AssertTrue(
    Condition := fb.sts.clampedHigh,
    Message   := 'Raw above rawMax must set clampedHigh');
AssertTrue(
    Condition := fb.sts.clampActive,
    Message   := 'clampActive must be TRUE when clampedHigh is set');
AssertTrue(
    Condition := ABS(fb.sts.value - 100.0) < TOL,
    Message   := 'Clamped-high output must pin to euMax (100 %)');

TEST_FINISHED();
END_METHOD

METHOD ClampPromotesGoodQualityToClamped
VAR
    fb : TcForge.FB_AnalogInput;
END_VAR
TEST('ClampPromotesGoodQualityToClamped');

// When the raw input is clamping *and* inpQuality = GOOD, the FB must
// promote quality to CLAMPED to signal "reading is legal but pinned".
fb.inRaw.nInt := -1;
fb(inpQuality := TcForge.E_IO_Quality.GOOD);

AssertTrue(
    Condition := fb.sts.clampActive,
    Message   := 'Precondition: clampActive must be TRUE');
AssertEquals_DINT(
    Expected := TO_DINT(TcForge.E_IO_Quality.CLAMPED),
    Actual   := TO_DINT(fb.sts.quality),
    Message  := 'GOOD quality must be promoted to CLAMPED while clamping');

TEST_FINISHED();
END_METHOD

METHOD ClampAsFaultRaisesClampLow
VAR
    fb : TcForge.FB_AnalogInput;
END_VAR
TEST('ClampAsFaultRaisesClampLow');

fb.cfg.clampAsFault := TRUE;
fb.inRaw.nInt := -10;
fb(inpQuality := TcForge.E_IO_Quality.GOOD);

AssertTrue(
    Condition := fb.sts.header.faulted,
    Message   := 'clampAsFault + raw below RawMin must fault the device');
AssertEquals_DINT(
    Expected := TcForge.E_AnalogInput_Fault.ClampLow,
    Actual   := fb.sts.header.faultCode,
    Message  := 'Fault code must be ClampLow');

TEST_FINISHED();
END_METHOD

METHOD ClampAsFaultRaisesClampHigh
VAR
    fb : TcForge.FB_AnalogInput;
END_VAR
TEST('ClampAsFaultRaisesClampHigh');

fb.cfg.clampAsFault := TRUE;
fb.cfg.inputType    := __SYSTEM.TYPE_CLASS.TYPE_REAL;
fb.inRaw.fReal := 50000.0;
fb(inpQuality := TcForge.E_IO_Quality.GOOD);

AssertTrue(
    Condition := fb.sts.header.faulted,
    Message   := 'clampAsFault + raw above RawMax must fault the device');
AssertEquals_DINT(
    Expected := TcForge.E_AnalogInput_Fault.ClampHigh,
    Actual   := fb.sts.header.faultCode,
    Message  := 'Fault code must be ClampHigh');

TEST_FINISHED();
END_METHOD

METHOD BadConfigRaisesFaultOnFirstScan
VAR
    fb : TcForge.FB_AnalogInput;
END_VAR
TEST('BadConfigRaisesFaultOnFirstScan');

// BadConfig check runs once on the first scan. Set rawMin >= rawMax
// BEFORE the first cyclic call so the validation can latch _configBad.
fb.cfg.rawMin := 100.0;
fb.cfg.rawMax := 100.0;
fb(inpQuality := TcForge.E_IO_Quality.GOOD);

AssertTrue(
    Condition := fb.sts.header.faulted,
    Message   := 'rawMin >= rawMax must fault the device as BadConfig');
AssertEquals_DINT(
    Expected := TcForge.E_AnalogInput_Fault.BadConfig,
    Actual   := fb.sts.header.faultCode,
    Message  := 'Fault code must be BadConfig');

TEST_FINISHED();
END_METHOD

METHOD BadQualityHoldsLastRawReading
VAR
    fb          : TcForge.FB_AnalogInput;
    snapshotRaw : REAL;
END_VAR
TEST('BadQualityHoldsLastRawReading');

// Establish a good reading first.
fb.inRaw.nInt := 10000;
fb(inpQuality := TcForge.E_IO_Quality.GOOD);
snapshotRaw := fb.sts.rawReal;

// Flip quality to BAD and change the raw wire. The FB must discard the
// fresh value and hold the last-known-good raw reading.
fb.inRaw.nInt := 25000;
fb(inpQuality := TcForge.E_IO_Quality.BAD);

AssertTrue(
    Condition := ABS(fb.sts.rawReal - snapshotRaw) < TOL,
    Message   := 'BAD quality must hold rawReal at the last-known-good value');

TEST_FINISHED();
END_METHOD

METHOD InputTypeRealReadsRealMemberOfUnion
VAR
    fb : TcForge.FB_AnalogInput;
END_VAR
TEST('InputTypeRealReadsRealMemberOfUnion');

// Select the REAL UNION member and reconfigure scaling so raw == EU,
// then confirm the FB reads the REAL alias rather than some other
// reinterpretation of the same bytes.
fb.cfg.inputType := __SYSTEM.TYPE_CLASS.TYPE_REAL;
fb.cfg.rawMin    := 0.0;
fb.cfg.rawMax    := 100.0;
fb.cfg.euMin     := 0.0;
fb.cfg.euMax     := 100.0;

fb.inRaw.fReal := 42.5;
fb(inpQuality := TcForge.E_IO_Quality.GOOD);

AssertTrue(
    Condition := ABS(fb.sts.rawReal - 42.5) < TOL,
    Message   := 'TYPE_REAL must read inRaw.fReal directly into rawReal');
AssertTrue(
    Condition := ABS(fb.sts.value - 42.5) < TOL,
    Message   := 'Identity scaling must leave value equal to the raw REAL input');

TEST_FINISHED();
END_METHOD

METHOD QualityTagPropagatesToStatus
VAR
    fb : TcForge.FB_AnalogInput;
END_VAR
TEST('QualityTagPropagatesToStatus');

// The FB must echo inpQuality into sts.quality each cycle (subject to
// the clamp promotion covered by ClampPromotesGoodQualityToClamped).
fb.inRaw.nInt := 10000;
fb(inpQuality := TcForge.E_IO_Quality.GOOD);
AssertEquals_DINT(
    Expected := TO_DINT(TcForge.E_IO_Quality.GOOD),
    Actual   := TO_DINT(fb.sts.quality),
    Message  := 'quality must mirror inpQuality = GOOD when not clamping');

fb(inpQuality := TcForge.E_IO_Quality.UNKNOWN);
AssertEquals_DINT(
    Expected := TO_DINT(TcForge.E_IO_Quality.UNKNOWN),
    Actual   := TO_DINT(fb.sts.quality),
    Message  := 'quality must mirror inpQuality = UNKNOWN');

fb(inpQuality := TcForge.E_IO_Quality.BAD);
AssertEquals_DINT(
    Expected := TO_DINT(TcForge.E_IO_Quality.BAD),
    Actual   := TO_DINT(fb.sts.quality),
    Message  := 'quality must mirror inpQuality = BAD');

TEST_FINISHED();
END_METHOD

END_FUNCTION_BLOCK

// ---- Tests/FB_AnalogOutput_Test.TcPOU
// Tests exercise the public input/output and command contracts.
FUNCTION_BLOCK FB_AnalogOutput_Test EXTENDS TcUnit.FB_TestSuite
VAR CONSTANT
    TOL     : REAL := 1E-3;
    RAW_TOL : INT  := 1;
END_VAR

InitialStatusPublishesDefaults();
LinearScalingMapsEndpointsAndMidpoint();
ClampHighPinsCommandAndFlagsClampedHigh();
ClampLowPinsCommandAndFlagsClampedLow();
CommandedEchoesUnclampedRequest();
RawBypassSkipsClampAndScaling();
ClampAsFaultRaisesClampHigh();
ClampAsFaultRaisesClampLow();
BadConfigRaisesFaultOnFirstScan();
OutputTypeRealWritesRealUnionMember();
BadQualityHoldsLastWrittenUnion();
QualityTagPropagatesToStatus();
SetValueRejectedWhenSourceLockedToProg();
SetValueAcceptedFromProgWhenLocked();

METHOD InitialStatusPublishesDefaults
VAR
    fb : TcForge.FB_AnalogOutput;
END_VAR
TEST('InitialStatusPublishesDefaults');

// Default cfg: INT terminal, EU 0..100 % scaled into raw 0..32767,
// clampAsFault disabled. Before any SetValue the persistent command is
// zero, so the FB must publish a clean zero command with no clamp
// flags and no fault.
fb(inpQuality := TcForge.E_IO_Quality.GOOD);

AssertTrue(
    Condition := ABS(fb.sts.value) < TOL,
    Message   := 'Fresh instance must publish value = 0 for an unset command');
AssertTrue(
    Condition := ABS(fb.sts.commanded) < TOL,
    Message   := 'Fresh instance must publish commanded = 0');
AssertTrue(
    Condition := ABS(fb.sts.rawReal) < TOL,
    Message   := 'Fresh instance must publish rawReal = 0');
AssertFalse(
    Condition := fb.sts.clampActive,
    Message   := 'Zero command is inside [minCv, maxCv] so clampActive must be FALSE');
AssertFalse(
    Condition := fb.sts.header.faulted,
    Message   := 'Default cfg is valid so the first scan must not fault');

TEST_FINISHED();
END_METHOD

METHOD LinearScalingMapsEndpointsAndMidpoint
VAR
    fb  : TcForge.FB_AnalogOutput;
    rsp : TcForge.E_RpcMethodResponse;
END_VAR
TEST('LinearScalingMapsEndpointsAndMidpoint');

// Default cfg: EU 0..100 -> raw 0..32767. Verify the two endpoints and
// the midpoint land where the linear recurrence says they should,
// both in sts.rawReal (REAL) and in outRaw.nInt (after INT coercion).
//
//     rawReal = rawMin + (cmd - euMin)
//                             * (rawMax - rawMin)
//                             / (euMax - euMin)

rsp := fb.SetValue(rValue := 0.0);
fb(inpQuality := TcForge.E_IO_Quality.GOOD);
AssertTrue(
    Condition := ABS(fb.sts.rawReal - 0.0) < TOL,
    Message   := 'cmd = euMin must map to rawMin (0)');
AssertTrue(
    Condition := ABS(fb.outRaw.nInt) <= RAW_TOL,
    Message   := 'UNION INT alias must receive ~0 for a 0 %% command');

rsp := fb.SetValue(rValue := 100.0);
fb(inpQuality := TcForge.E_IO_Quality.GOOD);
AssertTrue(
    Condition := ABS(fb.sts.rawReal - 32767.0) < TOL,
    Message   := 'cmd = euMax must map to rawMax (32767)');
AssertTrue(
    Condition := ABS(fb.outRaw.nInt - 32767) <= RAW_TOL,
    Message   := 'UNION INT alias must receive ~32767 for a 100 %% command');

rsp := fb.SetValue(rValue := 50.0);
fb(inpQuality := TcForge.E_IO_Quality.GOOD);
AssertTrue(
    Condition := ABS(fb.sts.rawReal - 16383.5) < 0.01,
    Message   := 'cmd at midpoint must map to raw midpoint');
AssertTrue(
    Condition := ABS(fb.outRaw.nInt - 16384) <= RAW_TOL,
    Message   := 'UNION INT alias must receive the rounded midpoint raw');

TEST_FINISHED();
END_METHOD

METHOD ClampHighPinsCommandAndFlagsClampedHigh
VAR
    fb  : TcForge.FB_AnalogOutput;
    rsp : TcForge.E_RpcMethodResponse;
END_VAR
TEST('ClampHighPinsCommandAndFlagsClampedHigh');

// Drive a command above maxCv. clampedHigh must fire, clampActive must
// track, value must pin at maxCv, and the raw write must use the
// pinned value — not the unclamped request.
rsp := fb.SetValue(rValue := 150.0);
fb(inpQuality := TcForge.E_IO_Quality.GOOD);

AssertTrue(
    Condition := fb.sts.clampedHigh,
    Message   := 'cmd above maxCv must set clampedHigh');
AssertTrue(
    Condition := fb.sts.clampActive,
    Message   := 'clampActive must be TRUE whenever either clamp direction is active');
AssertTrue(
    Condition := ABS(fb.sts.value - 100.0) < TOL,
    Message   := 'value must pin at maxCv (100 %%) when clamping high');
AssertTrue(
    Condition := ABS(fb.sts.rawReal - 32767.0) < TOL,
    Message   := 'rawReal must reflect the clamped EU, not the unclamped request');
AssertFalse(
    Condition := fb.sts.header.faulted,
    Message   := 'clampAsFault = FALSE by default; clamp alone must not fault the device');

TEST_FINISHED();
END_METHOD

METHOD ClampLowPinsCommandAndFlagsClampedLow
VAR
    fb  : TcForge.FB_AnalogOutput;
    rsp : TcForge.E_RpcMethodResponse;
END_VAR
TEST('ClampLowPinsCommandAndFlagsClampedLow');

// Drive a command below minCv. clampedLow must fire, value must pin
// at minCv, raw write uses the pinned value.
rsp := fb.SetValue(rValue := -25.0);
fb(inpQuality := TcForge.E_IO_Quality.GOOD);

AssertTrue(
    Condition := fb.sts.clampedLow,
    Message   := 'cmd below minCv must set clampedLow');
AssertTrue(
    Condition := fb.sts.clampActive,
    Message   := 'clampActive must be TRUE whenever either clamp direction is active');
AssertTrue(
    Condition := ABS(fb.sts.value - 0.0) < TOL,
    Message   := 'value must pin at minCv (0 %%) when clamping low');
AssertTrue(
    Condition := ABS(fb.sts.rawReal - 0.0) < TOL,
    Message   := 'rawReal must reflect the clamped EU, not the unclamped request');
AssertFalse(
    Condition := fb.sts.header.faulted,
    Message   := 'clampAsFault = FALSE by default; clamp alone must not fault the device');

TEST_FINISHED();
END_METHOD

METHOD CommandedEchoesUnclampedRequest
VAR
    fb  : TcForge.FB_AnalogOutput;
    rsp : TcForge.E_RpcMethodResponse;
END_VAR
TEST('CommandedEchoesUnclampedRequest');

// sts.commanded publishes the pre-clamp request; restart restoration is separately qualified
// via _requestSync. The tests above already prove sts.value tracks the
// clamped write; here we pin down that sts.commanded preserves the
// operator's original intent so the HMI can show "you asked for 150,
// we clamped to 100".
rsp := fb.SetValue(rValue := 150.0);
fb(inpQuality := TcForge.E_IO_Quality.GOOD);

AssertTrue(
    Condition := ABS(fb.sts.commanded - 150.0) < TOL,
    Message   := 'commanded must echo the unclamped SetValue input');
AssertTrue(
    Condition := ABS(fb.sts.value - 100.0) < TOL,
    Message   := 'value must be the clamped command actually written');

rsp := fb.SetValue(rValue := -7.5);
fb(inpQuality := TcForge.E_IO_Quality.GOOD);

AssertTrue(
    Condition := ABS(fb.sts.commanded - (-7.5)) < TOL,
    Message   := 'commanded must echo a negative request even when clamped low');
AssertTrue(
    Condition := ABS(fb.sts.value - 0.0) < TOL,
    Message   := 'value must pin at minCv under a low clamp');

TEST_FINISHED();
END_METHOD

METHOD RawBypassSkipsClampAndScaling
VAR
    fb  : TcForge.FB_AnalogOutput;
    rsp : TcForge.E_RpcMethodResponse;
END_VAR
TEST('RawBypassSkipsClampAndScaling');

// useRawValue = TRUE writes the command REAL straight into the UNION
// without clamping, so a 12345 command lands as 12345 on the raw INT
// alias even though that is well above maxCv and well above rawMax.
fb.cfg.useRawValue := TRUE;
rsp := fb.SetValue(rValue := 12345.0);
fb(inpQuality := TcForge.E_IO_Quality.GOOD);

AssertTrue(
    Condition := ABS(fb.sts.rawReal - 12345.0) < TOL,
    Message   := 'With useRawValue = TRUE, rawReal must equal the raw command');
AssertTrue(
    Condition := ABS(fb.sts.value - 12345.0) < TOL,
    Message   := 'With useRawValue = TRUE, value must equal the raw command');
AssertFalse(
    Condition := fb.sts.clampedLow,
    Message   := 'Raw bypass must not flag clampedLow');
AssertFalse(
    Condition := fb.sts.clampedHigh,
    Message   := 'Raw bypass must not flag clampedHigh');
AssertFalse(
    Condition := fb.sts.clampActive,
    Message   := 'Raw bypass must not flag clampActive');
AssertTrue(
    Condition := ABS(fb.outRaw.nInt - 12345) <= RAW_TOL,
    Message   := 'UNION INT alias must receive the raw command unchanged');

TEST_FINISHED();
END_METHOD

METHOD ClampAsFaultRaisesClampHigh
VAR
    fb  : TcForge.FB_AnalogOutput;
    rsp : TcForge.E_RpcMethodResponse;
END_VAR
TEST('ClampAsFaultRaisesClampHigh');

fb.cfg.clampAsFault := TRUE;
rsp := fb.SetValue(rValue := 150.0);
fb(inpQuality := TcForge.E_IO_Quality.GOOD);

AssertTrue(
    Condition := fb.sts.header.faulted,
    Message   := 'clampAsFault + cmd above maxCv must fault the device');
AssertEquals_DINT(
    Expected := TcForge.E_AnalogOutput_Fault.ClampHigh,
    Actual   := fb.sts.header.faultCode,
    Message  := 'Fault code must be ClampHigh');

TEST_FINISHED();
END_METHOD

METHOD ClampAsFaultRaisesClampLow
VAR
    fb  : TcForge.FB_AnalogOutput;
    rsp : TcForge.E_RpcMethodResponse;
END_VAR
TEST('ClampAsFaultRaisesClampLow');

fb.cfg.clampAsFault := TRUE;
rsp := fb.SetValue(rValue := -5.0);
fb(inpQuality := TcForge.E_IO_Quality.GOOD);

AssertTrue(
    Condition := fb.sts.header.faulted,
    Message   := 'clampAsFault + cmd below minCv must fault the device');
AssertEquals_DINT(
    Expected := TcForge.E_AnalogOutput_Fault.ClampLow,
    Actual   := fb.sts.header.faultCode,
    Message  := 'Fault code must be ClampLow');

TEST_FINISHED();
END_METHOD

METHOD BadConfigRaisesFaultOnFirstScan
VAR
    fb : TcForge.FB_AnalogOutput;
END_VAR
TEST('BadConfigRaisesFaultOnFirstScan');

// BadConfig check runs once on the first scan. Set rawMin > rawMax
// BEFORE the first cyclic call so the validation can latch _configBad.
fb.cfg.rawMin := 200.0;
fb.cfg.rawMax := 100.0;
fb(inpQuality := TcForge.E_IO_Quality.GOOD);

AssertTrue(
    Condition := fb.sts.header.faulted,
    Message   := 'rawMin > rawMax must fault the device as BadConfig');
AssertEquals_DINT(
    Expected := TcForge.E_AnalogOutput_Fault.BadConfig,
    Actual   := fb.sts.header.faultCode,
    Message  := 'Fault code must be BadConfig');

TEST_FINISHED();
END_METHOD

METHOD OutputTypeRealWritesRealUnionMember
VAR
    fb  : TcForge.FB_AnalogOutput;
    rsp : TcForge.E_RpcMethodResponse;
END_VAR
TEST('OutputTypeRealWritesRealUnionMember');

// Select the REAL UNION member and reconfigure scaling so raw == EU,
// then confirm the FB writes the REAL alias with the exact command
// (no integer coercion).
fb.cfg.outputType := __SYSTEM.TYPE_CLASS.TYPE_REAL;
fb.cfg.rawMin     := 0.0;
fb.cfg.rawMax     := 100.0;
fb.cfg.euMin      := 0.0;
fb.cfg.euMax      := 100.0;

rsp := fb.SetValue(rValue := 42.5);
fb(inpQuality := TcForge.E_IO_Quality.GOOD);

AssertTrue(
    Condition := ABS(fb.sts.rawReal - 42.5) < TOL,
    Message   := 'Identity scaling must leave rawReal equal to the command');
AssertTrue(
    Condition := ABS(fb.outRaw.fReal - 42.5) < TOL,
    Message   := 'TYPE_REAL must write outRaw.fReal directly with the command');

TEST_FINISHED();
END_METHOD

METHOD BadQualityHoldsLastWrittenUnion
VAR
    fb           : TcForge.FB_AnalogOutput;
    rsp          : TcForge.E_RpcMethodResponse;
    snapshot     : DWORD;
END_VAR
TEST('BadQualityHoldsLastWrittenUnion');
fb.cfg.holdOnBadQuality := TRUE;

// Establish a known value in the UNION under GOOD quality.
rsp := fb.SetValue(rValue := 25.0);
fb(inpQuality := TcForge.E_IO_Quality.GOOD);
snapshot := fb.outRaw.dw;

// Flip quality to BAD and change the commanded value. The FB must
// still recompute sts.rawReal (it is pure output of the pipeline),
// but it must NOT touch the hardware-linked UNION — the terminal
// keeps its last-known-good bytes.
rsp := fb.SetValue(rValue := 75.0);
fb(inpQuality := TcForge.E_IO_Quality.BAD);

AssertEquals_DWORD(
    Expected := snapshot,
    Actual   := fb.outRaw.dw,
    Message  := 'BAD quality must skip the UNION write and hold the last-known-good bytes');

TEST_FINISHED();
END_METHOD

METHOD QualityTagPropagatesToStatus
VAR
    fb : TcForge.FB_AnalogOutput;
END_VAR
TEST('QualityTagPropagatesToStatus');

// FB_AnalogOutput echoes inpQuality straight through (no clamp-to-CLAMPED
// promotion like the input FB does — output-side consumers treat CLAMPED
// as informational and the write still goes out).
fb(inpQuality := TcForge.E_IO_Quality.GOOD);
AssertEquals_DINT(
    Expected := TO_DINT(TcForge.E_IO_Quality.GOOD),
    Actual   := TO_DINT(fb.sts.quality),
    Message  := 'quality must mirror inpQuality = GOOD');

fb(inpQuality := TcForge.E_IO_Quality.UNKNOWN);
AssertEquals_DINT(
    Expected := TO_DINT(TcForge.E_IO_Quality.UNKNOWN),
    Actual   := TO_DINT(fb.sts.quality),
    Message  := 'quality must mirror inpQuality = UNKNOWN');

fb(inpQuality := TcForge.E_IO_Quality.BAD);
AssertEquals_DINT(
    Expected := TO_DINT(TcForge.E_IO_Quality.BAD),
    Actual   := TO_DINT(fb.sts.quality),
    Message  := 'quality must mirror inpQuality = BAD');

TEST_FINISHED();
END_METHOD

METHOD SetValueRejectedWhenSourceLockedToProg
VAR
    fb  : TcForge.FB_AnalogOutput;
    rsp : TcForge.E_RpcMethodResponse;
END_VAR
TEST('SetValueRejectedWhenSourceLockedToProg');

// With source locked to PROG, an OPERATOR SetValue must be rejected
// with SOURCE_LOCKED, the persistent command must stay at zero, and
// no clamp flags or writes may trigger.
fb.LockSource(bLock := TRUE);

rsp := fb.SetValue(rValue := 42.0, eRequester := TcForge.E_Requester.OPERATOR);
fb(inpQuality := TcForge.E_IO_Quality.GOOD);

AssertEquals_DINT(
    Expected := TO_DINT(TcForge.E_RpcMethodResponse.REJECTED_SOURCE_NOT_ALLOWED),
    Actual   := TO_DINT(rsp),
    Message  := 'OPERATOR SetValue against a source-locked FB must be rejected');
AssertTrue(
    Condition := ABS(fb.sts.commanded - 0.0) < TOL,
    Message   := 'A rejected SetValue must leave commanded unchanged');
AssertTrue(
    Condition := ABS(fb.sts.value - 0.0) < TOL,
    Message   := 'A rejected SetValue must leave value unchanged');

TEST_FINISHED();
END_METHOD

METHOD SetValueAcceptedFromProgWhenLocked
VAR
    fb  : TcForge.FB_AnalogOutput;
    rsp : TcForge.E_RpcMethodResponse;
END_VAR
TEST('SetValueAcceptedFromProgWhenLocked');

// With source locked to PROG, a PROG SetValue must still be accepted —
// that's the whole point of locking: only the program may drive.
fb.LockSource(bLock := TRUE);

rsp := fb.SetValue(rValue := 42.0, eRequester := TcForge.E_Requester.PROG);
fb(inpQuality := TcForge.E_IO_Quality.GOOD);

AssertEquals_DINT(
    Expected := TO_DINT(TcForge.E_RpcMethodResponse.ACCEPTED),
    Actual   := TO_DINT(rsp),
    Message  := 'PROG SetValue must be accepted even when source-locked to PROG');
AssertTrue(
    Condition := ABS(fb.sts.commanded - 42.0) < TOL,
    Message   := 'Accepted PROG SetValue must update commanded');
AssertTrue(
    Condition := ABS(fb.sts.value - 42.0) < TOL,
    Message   := 'Accepted PROG SetValue must flow into value');

TEST_FINISHED();
END_METHOD

END_FUNCTION_BLOCK

// ---- Tests/FB_AlarmThreshold_Test.TcPOU
// Tests for FB_AlarmThreshold. The FB itself is thin — it owns the
// direction select (bFailHigh / bFailLow) and the raw comparator, then
// forwards everything into FB_AlarmBase._Evaluate(). The shared alarm
// contract (debounce, latch/ack state machine, severity, message echo,
// source lock, disable gating) is already covered by FB_AlarmSimple_Test,
// so this suite focuses on the threshold-specific logic plus a couple of
// smoke tests that confirm the base pipeline is wired in.
FUNCTION_BLOCK FB_AlarmThreshold_Test EXTENDS TcUnit.FB_TestSuite

FailHighTripsStrictlyAboveThreshold();
FailHighIgnoresAtOrBelowThreshold();
FailLowTripsStrictlyBelowThreshold();
FailLowIgnoresAtOrAboveThreshold();
BothDirectionsAreInvalid();
NeitherDirectionIsInvalid();
DisabledSuppressesTripRegardlessOfValue();
SeverityFlowsThroughBaseOnActive();
LatchingHoldsAfterValueReturnsToSafe();
MessageEchoedFromCommonCfg();

METHOD FailHighTripsStrictlyAboveThreshold
VAR
    fb : TcForge.FB_AlarmThreshold;
END_VAR
TEST('FailHighTripsStrictlyAboveThreshold');

// bFailHigh + inpValue > fThreshold must trip the alarm. Configured as
// non-latching so we can observe the raw rollup directly.
fb.cfg.common.bEnable := TRUE;
fb.cfg.fThreshold     := 80.0;
fb.cfg.bFailHigh      := TRUE;

fb(inpValue := 80.1);
AssertTrue(
    Condition := fb.sts.active,
    Message   := 'Fail-high alarm must go active when inpValue exceeds fThreshold');
AssertTrue(
    Condition := fb.sts.raw,
    Message   := 'Fail-high rollup must mirror the strict > comparison on sts.raw');

TEST_FINISHED();
END_METHOD

METHOD FailHighIgnoresAtOrBelowThreshold
VAR
    fb : TcForge.FB_AlarmThreshold;
END_VAR
TEST('FailHighIgnoresAtOrBelowThreshold');

// inpValue == fThreshold must NOT trip a fail-high alarm: the comparison
// is a strict `>` so a reading that is exactly at the threshold is
// considered still-safe. Any inequality in the other direction is also
// ignored. Together these prevent jittery readings from chattering on
// the threshold boundary.
fb.cfg.common.bEnable := TRUE;
fb.cfg.fThreshold     := 80.0;
fb.cfg.bFailHigh      := TRUE;

fb(inpValue := 80.0);
AssertFalse(
    Condition := fb.sts.active,
    Message   := 'Fail-high must not trip when inpValue equals fThreshold (strict >)');

fb(inpValue := 10.0);
AssertFalse(
    Condition := fb.sts.active,
    Message   := 'Fail-high must not trip when inpValue is well below fThreshold');

TEST_FINISHED();
END_METHOD

METHOD FailLowTripsStrictlyBelowThreshold
VAR
    fb : TcForge.FB_AlarmThreshold;
END_VAR
TEST('FailLowTripsStrictlyBelowThreshold');

fb.cfg.common.bEnable := TRUE;
fb.cfg.fThreshold     := 10.0;
fb.cfg.bFailLow       := TRUE;

fb(inpValue := 9.9);
AssertTrue(
    Condition := fb.sts.active,
    Message   := 'Fail-low alarm must go active when inpValue falls below fThreshold');

TEST_FINISHED();
END_METHOD

METHOD FailLowIgnoresAtOrAboveThreshold
VAR
    fb : TcForge.FB_AlarmThreshold;
END_VAR
TEST('FailLowIgnoresAtOrAboveThreshold');

fb.cfg.common.bEnable := TRUE;
fb.cfg.fThreshold     := 10.0;
fb.cfg.bFailLow       := TRUE;

fb(inpValue := 10.0);
AssertFalse(
    Condition := fb.sts.active,
    Message   := 'Fail-low must not trip when inpValue equals fThreshold (strict <)');

fb(inpValue := 50.0);
AssertFalse(
    Condition := fb.sts.active,
    Message   := 'Fail-low must not trip when inpValue is well above fThreshold');

TEST_FINISHED();
END_METHOD

METHOD BothDirectionsAreInvalid
VAR
    fb : TcForge.FB_AlarmThreshold;
END_VAR
TEST('BothDirectionsAreInvalid');
fb.cfg.common.bEnable := TRUE;
fb.cfg.bFailHigh := TRUE; fb.cfg.bFailLow := TRUE;
fb(inpValue := 60.0);
AssertFalse(Condition := fb.sts.valid, Message := 'Exactly one direction is required');
AssertEquals_DINT(Expected := TcForge.E_AlarmEvaluation.InvalidConfig, Actual := fb.sts.evaluationState, Message := 'Invalid configuration is visible');
AssertFalse(Condition := fb.sts.active, Message := 'Invalid fresh configuration does not invent a trip');
TEST_FINISHED();
END_METHOD

METHOD NeitherDirectionIsInvalid
VAR
    fb : TcForge.FB_AlarmThreshold;
END_VAR
TEST('NeitherDirectionIsInvalid');
fb.cfg.common.bEnable := TRUE;
fb.cfg.bFailHigh := FALSE; fb.cfg.bFailLow := FALSE;
fb(inpValue := 60.0);
AssertFalse(Condition := fb.sts.valid, Message := 'Exactly one direction is required');
AssertEquals_DINT(Expected := TcForge.E_AlarmEvaluation.InvalidConfig, Actual := fb.sts.evaluationState, Message := 'Invalid configuration is visible');
AssertFalse(Condition := fb.sts.active, Message := 'Invalid fresh configuration does not invent a trip');
TEST_FINISHED();
END_METHOD

METHOD DisabledSuppressesTripRegardlessOfValue
VAR
    fb : TcForge.FB_AlarmThreshold;
END_VAR
TEST('DisabledSuppressesTripRegardlessOfValue');

// bEnable = FALSE shortcuts _Evaluate before the latch / severity logic
// runs. Confirm the threshold FB inherits that behaviour even when the
// raw comparison would otherwise fire.
fb.cfg.common.bEnable := FALSE;
fb.cfg.common.eSeverity := TcForge.E_AlarmSeverity.CRITICAL;
fb.cfg.fThreshold       := 50.0;
fb.cfg.bFailHigh        := TRUE;

fb(inpValue := 999.0);

AssertFalse(
    Condition := fb.sts.active,
    Message   := 'Disabled threshold alarm must not trip even with inpValue way above fThreshold');
AssertEquals_USINT(
    Expected := TcForge.E_AlarmSeverity.NONE,
    Actual   := fb.sts.eSeverity,
    Message  := 'Disabled alarm must report severity NONE regardless of value');

TEST_FINISHED();
END_METHOD

METHOD SeverityFlowsThroughBaseOnActive
VAR
    fb : TcForge.FB_AlarmThreshold;
END_VAR
TEST('SeverityFlowsThroughBaseOnActive');

// Smoke test: when the threshold condition trips, the base's severity
// propagation still runs. This proves the threshold FB does call
// _Evaluate() and does not short-circuit the pipeline.
fb.cfg.common.bEnable     := TRUE;
fb.cfg.common.bRequireAck := FALSE;
fb.cfg.common.eSeverity   := TcForge.E_AlarmSeverity.WARNING;
fb.cfg.fThreshold         := 50.0;
fb.cfg.bFailHigh          := TRUE;

fb(inpValue := 60.0);
AssertEquals_USINT(
    Expected := TcForge.E_AlarmSeverity.WARNING,
    Actual   := fb.sts.eSeverity,
    Message  := 'Active threshold alarm must publish the configured severity');

fb(inpValue := 40.0);
AssertEquals_USINT(
    Expected := TcForge.E_AlarmSeverity.NONE,
    Actual   := fb.sts.eSeverity,
    Message  := 'Cleared threshold alarm must drop severity to NONE');

TEST_FINISHED();
END_METHOD

METHOD LatchingHoldsAfterValueReturnsToSafe
VAR
    fb : TcForge.FB_AlarmThreshold;
END_VAR
TEST('LatchingHoldsAfterValueReturnsToSafe');

// Smoke test for the bRequireAck pathway through the threshold FB.
// The base FB_AlarmSimple_Test already exercises the full latch/ack
// state machine in isolation; here we just confirm the threshold FB
// keeps the latch engaged after the process value returns below the
// threshold (which is the whole reason to latch on a transient spike).
fb.cfg.common.bEnable     := TRUE;
fb.cfg.common.bRequireAck := TRUE;
fb.cfg.common.eSeverity   := TcForge.E_AlarmSeverity.CRITICAL;
fb.cfg.fThreshold         := 80.0;
fb.cfg.bFailHigh          := TRUE;

fb(inpValue := 90.0);
AssertTrue(
    Condition := fb.sts.active AND fb.sts.latched,
    Message   := 'Latching threshold alarm must go active+latched on a trip');

fb(inpValue := 50.0);
AssertTrue(
    Condition := fb.sts.active,
    Message   := 'Latched threshold alarm must stay active after inpValue returns below fThreshold');

TEST_FINISHED();
END_METHOD

METHOD MessageEchoedFromCommonCfg
VAR
    fb : TcForge.FB_AlarmThreshold;
END_VAR
TEST('MessageEchoedFromCommonCfg');

// Confirms that a threshold alarm hands the common cfg (including
// sMessage) to the base unchanged. Regression guard against future
// refactors of ST_AlarmThreshold_Cfg that might shadow `common`.
fb.cfg.common.bEnable  := TRUE;
fb.cfg.common.sMessage := 'Reactor temp > 80C';
fb.cfg.fThreshold      := 80.0;
fb.cfg.bFailHigh       := TRUE;

fb(inpValue := 50.0);

AssertEquals_STRING(
    Expected := 'Reactor temp > 80C',
    Actual   := fb.sts.sMessage,
    Message  := 'sts.sMessage must echo cfg.common.sMessage verbatim');

TEST_FINISHED();
END_METHOD

END_FUNCTION_BLOCK

// ---- Tests/FB_AlarmDeviation_Test.TcPOU
// Tests for FB_AlarmDeviation. The deviation FB owns two comparator
// modes — absolute band (fLowLimit..fHighLimit) and asymmetric setpoint
// deviation (inpSetpoint +/- limit) — and forwards the boolean rollup
// into FB_AlarmBase._Evaluate(). The shared alarm contract (debounce,
// latch/ack, severity, source lock) is already covered by
// FB_AlarmSimple_Test, so this suite focuses on the deviation-specific
// comparator logic plus a smoke test confirming the base pipeline runs.
FUNCTION_BLOCK FB_AlarmDeviation_Test EXTENDS TcUnit.FB_TestSuite

AbsoluteModeTripsAboveHighLimit();
AbsoluteModeTripsBelowLowLimit();
AbsoluteModeStaysQuietWithinBand();
AbsoluteModeIgnoresInpSetpoint();
SetpointModeTripsAbovePositiveDeviation();
SetpointModeTripsBelowNegativeDeviation();
SetpointModeTracksMovingSetpoint();
SetpointModeAllowsAsymmetricLimits();
DisabledSuppressesTripRegardlessOfValue();
SeverityFlowsThroughBaseOnActive();

METHOD AbsoluteModeTripsAboveHighLimit
VAR
    fb : TcForge.FB_AlarmDeviation;
END_VAR
TEST('AbsoluteModeTripsAboveHighLimit');

// Absolute mode: limits are direct values on inpPv (inpSetpoint ignored).
fb.cfg.common.bEnable := TRUE;
fb.cfg.bUseSetpoint   := FALSE;
fb.cfg.fHighLimit     := 95.0;
fb.cfg.fLowLimit      := 10.0;

fb(inpPv := 96.0, inpSetpoint := 0.0);

AssertTrue(
    Condition := fb.sts.active,
    Message   := 'Absolute mode must trip when inpPv is strictly above fHighLimit');

TEST_FINISHED();
END_METHOD

METHOD AbsoluteModeTripsBelowLowLimit
VAR
    fb : TcForge.FB_AlarmDeviation;
END_VAR
TEST('AbsoluteModeTripsBelowLowLimit');

fb.cfg.common.bEnable := TRUE;
fb.cfg.bUseSetpoint   := FALSE;
fb.cfg.fHighLimit     := 95.0;
fb.cfg.fLowLimit      := 10.0;

fb(inpPv := 9.0, inpSetpoint := 0.0);

AssertTrue(
    Condition := fb.sts.active,
    Message   := 'Absolute mode must trip when inpPv is strictly below fLowLimit');

TEST_FINISHED();
END_METHOD

METHOD AbsoluteModeStaysQuietWithinBand
VAR
    fb : TcForge.FB_AlarmDeviation;
END_VAR
TEST('AbsoluteModeStaysQuietWithinBand');

// Boundaries are inclusive (strict > and strict <), so exactly-at-limit
// readings must not trip. Middle-of-band must also not trip.
fb.cfg.common.bEnable := TRUE;
fb.cfg.bUseSetpoint   := FALSE;
fb.cfg.fHighLimit     := 95.0;
fb.cfg.fLowLimit      := 10.0;

fb(inpPv := 10.0);
AssertFalse(
    Condition := fb.sts.active,
    Message   := 'Absolute mode must not trip at the low boundary exactly (strict <)');

fb(inpPv := 95.0);
AssertFalse(
    Condition := fb.sts.active,
    Message   := 'Absolute mode must not trip at the high boundary exactly (strict >)');

fb(inpPv := 50.0);
AssertFalse(
    Condition := fb.sts.active,
    Message   := 'Absolute mode must not trip mid-band');

TEST_FINISHED();
END_METHOD

METHOD AbsoluteModeIgnoresInpSetpoint
VAR
    fb : TcForge.FB_AlarmDeviation;
END_VAR
TEST('AbsoluteModeIgnoresInpSetpoint');

// Absolute mode must not look at inpSetpoint at all — otherwise a drifting
// setpoint could silently shift the safe band. Same PV, different SP,
// same result.
fb.cfg.common.bEnable := TRUE;
fb.cfg.bUseSetpoint   := FALSE;
fb.cfg.fHighLimit     := 95.0;
fb.cfg.fLowLimit      := 10.0;

fb(inpPv := 50.0, inpSetpoint := 0.0);
AssertFalse(
    Condition := fb.sts.active,
    Message   := 'Absolute mode with SP=0: mid-band must stay quiet');

fb(inpPv := 50.0, inpSetpoint := 1000.0);
AssertFalse(
    Condition := fb.sts.active,
    Message   := 'Absolute mode must ignore inpSetpoint: same PV stays quiet regardless of SP');

TEST_FINISHED();
END_METHOD

METHOD SetpointModeTripsAbovePositiveDeviation
VAR
    fb : TcForge.FB_AlarmDeviation;
END_VAR
TEST('SetpointModeTripsAbovePositiveDeviation');

// Setpoint mode: fHighLimit is a +deviation from inpSetpoint.
// SP=100, +5 band => trip above 105.
fb.cfg.common.bEnable := TRUE;
fb.cfg.bUseSetpoint   := TRUE;
fb.cfg.fHighLimit     := 5.0;
fb.cfg.fLowLimit      := 5.0;

fb(inpPv := 106.0, inpSetpoint := 100.0);

AssertTrue(
    Condition := fb.sts.active,
    Message   := 'Setpoint mode must trip when inpPv exceeds inpSetpoint + fHighLimit');

TEST_FINISHED();
END_METHOD

METHOD SetpointModeTripsBelowNegativeDeviation
VAR
    fb : TcForge.FB_AlarmDeviation;
END_VAR
TEST('SetpointModeTripsBelowNegativeDeviation');

fb.cfg.common.bEnable := TRUE;
fb.cfg.bUseSetpoint   := TRUE;
fb.cfg.fHighLimit     := 5.0;
fb.cfg.fLowLimit      := 5.0;

fb(inpPv := 94.0, inpSetpoint := 100.0);

AssertTrue(
    Condition := fb.sts.active,
    Message   := 'Setpoint mode must trip when inpPv falls below inpSetpoint - fLowLimit');

TEST_FINISHED();
END_METHOD

METHOD SetpointModeTracksMovingSetpoint
VAR
    fb : TcForge.FB_AlarmDeviation;
END_VAR
TEST('SetpointModeTracksMovingSetpoint');

// Whole point of setpoint mode: the safe band follows the setpoint.
// A PV that was in-band at SP=100 must be out-of-band once SP=200 if the
// deviations are small — and back in-band when SP catches up.
fb.cfg.common.bEnable     := TRUE;
fb.cfg.common.bRequireAck := FALSE;
fb.cfg.bUseSetpoint       := TRUE;
fb.cfg.fHighLimit         := 5.0;
fb.cfg.fLowLimit          := 5.0;

// PV=100 is dead on SP=100 => safe.
fb(inpPv := 100.0, inpSetpoint := 100.0);
AssertFalse(
    Condition := fb.sts.active,
    Message   := 'PV at SP is always safe');

// SP jumps to 200 before PV catches up => PV=100 is now 100 units low
// (well below SP-5 = 195) => trip.
fb(inpPv := 100.0, inpSetpoint := 200.0);
AssertTrue(
    Condition := fb.sts.active,
    Message   := 'SP jump away from PV must flip the deviation alarm active');

// PV catches up. Alarm clears next cycle since bRequireAck=FALSE.
fb(inpPv := 200.0, inpSetpoint := 200.0);
AssertFalse(
    Condition := fb.sts.active,
    Message   := 'PV catching up to SP must clear the deviation alarm');

TEST_FINISHED();
END_METHOD

METHOD SetpointModeAllowsAsymmetricLimits
VAR
    fb : TcForge.FB_AlarmDeviation;
END_VAR
TEST('SetpointModeAllowsAsymmetricLimits');

// Different tolerances above vs below the setpoint. Useful for processes
// where overshoot is dangerous but undershoot is fine (or vice versa).
// +10 allowed above, only -1 below.
fb.cfg.common.bEnable := TRUE;
fb.cfg.bUseSetpoint   := TRUE;
fb.cfg.fHighLimit     := 10.0;
fb.cfg.fLowLimit      := 1.0;

// SP=50, PV=58 is +8 => inside +10 band, no trip.
fb(inpPv := 58.0, inpSetpoint := 50.0);
AssertFalse(
    Condition := fb.sts.active,
    Message   := 'PV within the asymmetric high band (+8 of +10) must not trip');

// SP=50, PV=48 is -2 => below -1 band, trip.
fb(inpPv := 48.0, inpSetpoint := 50.0);
AssertTrue(
    Condition := fb.sts.active,
    Message   := 'PV outside the tight low band (-2 vs -1) must trip');

TEST_FINISHED();
END_METHOD

METHOD DisabledSuppressesTripRegardlessOfValue
VAR
    fb : TcForge.FB_AlarmDeviation;
END_VAR
TEST('DisabledSuppressesTripRegardlessOfValue');

fb.cfg.common.bEnable   := FALSE;
fb.cfg.common.eSeverity := TcForge.E_AlarmSeverity.CRITICAL;
fb.cfg.bUseSetpoint     := TRUE;
fb.cfg.fHighLimit       := 5.0;
fb.cfg.fLowLimit        := 5.0;

fb(inpPv := 1000.0, inpSetpoint := 0.0);

AssertFalse(
    Condition := fb.sts.active,
    Message   := 'Disabled deviation alarm must not trip even with extreme PV');
AssertEquals_USINT(
    Expected := TcForge.E_AlarmSeverity.NONE,
    Actual   := fb.sts.eSeverity,
    Message  := 'Disabled alarm must report severity NONE');

TEST_FINISHED();
END_METHOD

METHOD SeverityFlowsThroughBaseOnActive
VAR
    fb : TcForge.FB_AlarmDeviation;
END_VAR
TEST('SeverityFlowsThroughBaseOnActive');

// Smoke test: proves the deviation FB calls _Evaluate() so severity
// propagation works through the base pipeline.
fb.cfg.common.bEnable     := TRUE;
fb.cfg.common.bRequireAck := FALSE;
fb.cfg.common.eSeverity   := TcForge.E_AlarmSeverity.WARNING;
fb.cfg.bUseSetpoint       := FALSE;
fb.cfg.fHighLimit         := 50.0;
fb.cfg.fLowLimit          := 0.0;

fb(inpPv := 60.0);
AssertEquals_USINT(
    Expected := TcForge.E_AlarmSeverity.WARNING,
    Actual   := fb.sts.eSeverity,
    Message  := 'Active deviation alarm must publish the configured severity');

fb(inpPv := 25.0);
AssertEquals_USINT(
    Expected := TcForge.E_AlarmSeverity.NONE,
    Actual   := fb.sts.eSeverity,
    Message  := 'Cleared deviation alarm must drop severity to NONE');

TEST_FINISHED();
END_METHOD

END_FUNCTION_BLOCK

// ---- Tests/FB_Step_Test.TcPOU
// Tests for FB_Step, the lightweight step-lifecycle wrapper used inside
// FB_StateMachine sequences. FB_Step only reports "am I active?" and
// drives Entry / Execute / Exiting / Advance on top of the parent SM.
//
// Test strategy: FB_Step reads sm.Status.Step.Current via VAR_IN_OUT to
// decide whether it is the active step. Status is a VAR_OUTPUT on the
// production FB, which TwinCAT makes read-only from outside, so we
// drive activation via an FB_StateMachine_Probe that exposes a narrow
// SetCurrentStep / SetTimerSeconds pair and skips the parent body. The
// SM body is never called here — the tests observe FB_Step's own outputs
// (Entry/Execute/Exiting), the Step.Name it publishes, and the inherited
// fault book-keeping (sm.GetFaultCode()). End-to-end sequencing through
// the full SM body belongs in a separate FB_StateMachine suite.
//
// Shared-sm note: FB_StateMachine is a heavyweight FB (~35 KB, four
// FB_Permissives + an FB_Interlock + a full ST_SM_Status). TwinCAT
// places method-local VAR on the task stack (default 48 KB), so one
// probe per method blew the stack (C0297) and crashed the runtime
// during activation. We therefore share a single probe on the suite
// FB and reset it between tests via Setup(). `step : FB_Step` stays
// method-local — each test gets its own fresh lifecycle state, which
// is what makes the Entry/Execute/Exiting one-shots observable.
FUNCTION_BLOCK FB_Step_Test EXTENDS TcUnit.FB_TestSuite
VAR
    sm : FB_StateMachine_Probe;
END_VAR

InactiveKeepsLifecycleOutputsClear();
EntryRaisedOnFirstActiveScan();
ExecuteRaisedOnSecondActiveScanForPermSettle();
ExitingFiresOneShotAfterPermsAutoSatisfied();
AdvancePhaseKeepsAllLifecycleOutputsClear();
NamePublishedIntoSmStepInfo();
MappedFalsePermHoldsExecuteAndBlocksExit();
MappedTruePermLetsExitFireAfterSettle();
ZeroTimeoutNeverRaisesTimeoutFault();
TimeoutRaisesStepTimeoutFault();
InactiveRaiseFaultIsNoOp();
RaiseFaultWhileActiveRecordsCode();

// Prepare the shared SM probe for the next test. Reset the fault
// book-keeping, zero the timer, and force Step.Current to something
// the step-under-test will treat as inactive. The test then flips
// Step.Current to its own nStep so step sees a clean FALSE -> TRUE
// transition and Entry fires on the first call.
METHOD PRIVATE Setup
VAR
    rsp : TcForge.E_RpcMethodResponse;
END_VAR
sm.ResetAll();
sm.ForceState(state := TcForge.E_SM_State.RUNNING);
sm.SetCurrentStep(nStep := 9999);
sm.SetTimerSeconds(seconds := 0.0);
END_METHOD

METHOD InactiveKeepsLifecycleOutputsClear
VAR
    step : TcForge.FB_Step;
END_VAR
TEST('InactiveKeepsLifecycleOutputsClear');

// Baseline sanity: while the SM is advertising a different step,
// FB_Step must keep every lifecycle output FALSE and must not publish
// anything into Step.Name (a stale name would confuse the HMI).
Setup();

step(sm := sm, nStep := 3000, nNextStep := 3002, nTimeout := 0, sName := 'Inactive');

AssertFalse(
    Condition := step.Entry,
    Message   := 'Entry must be FALSE while the step is not the active one');
AssertFalse(
    Condition := step.Execute,
    Message   := 'Execute must be FALSE while the step is not the active one');
AssertFalse(
    Condition := step.Exiting,
    Message   := 'Exiting must be FALSE while the step is not the active one');

TEST_FINISHED();
END_METHOD

METHOD EntryRaisedOnFirstActiveScan
VAR
    step : TcForge.FB_Step;
END_VAR
TEST('EntryRaisedOnFirstActiveScan');

// First scan where _active flips FALSE -> TRUE must produce exactly one
// Entry pulse. Execute and Exiting must stay low so user init code
// (one-shot) runs without also running cyclic work on the same scan.
Setup();
sm.SetCurrentStep(nStep := 3000);

step(sm := sm, nStep := 3000, nNextStep := 3002, nTimeout := 0, sName := 'EntryScan');

AssertTrue(
    Condition := step.Entry,
    Message   := 'Entry must pulse TRUE on the first active scan');
AssertFalse(
    Condition := step.Execute,
    Message   := 'Execute must be FALSE on the Entry scan (no cyclic work yet)');
AssertFalse(
    Condition := step.Exiting,
    Message   := 'Exiting must be FALSE on the Entry scan');

TEST_FINISHED();
END_METHOD

METHOD ExecuteRaisedOnSecondActiveScanForPermSettle
VAR
    step : TcForge.FB_Step;
END_VAR
TEST('ExecuteRaisedOnSecondActiveScanForPermSettle');

// Second scan holds Execute high for one cycle even if no perms were
// mapped, so user MapPerm calls from the Entry scan get evaluated on
// the *next* scan before Exiting can fire. Without this settle, a step
// with no user work would skip Execute entirely.
Setup();
sm.SetCurrentStep(nStep := 3000);

step(sm := sm, nStep := 3000, nNextStep := 3002, nTimeout := 0, sName := 'Settle');
step(sm := sm, nStep := 3000, nNextStep := 3002, nTimeout := 0, sName := 'Settle');

AssertFalse(
    Condition := step.Entry,
    Message   := 'Entry must drop to FALSE after its one-shot Entry scan');
AssertTrue(
    Condition := step.Execute,
    Message   := 'Execute must fire on the second active scan (perm-settle pass)');
AssertFalse(
    Condition := step.Exiting,
    Message   := 'Exiting must not fire before the perm-settle pass has run');

TEST_FINISHED();
END_METHOD

METHOD ExitingFiresOneShotAfterPermsAutoSatisfied
VAR
    step : TcForge.FB_Step;
END_VAR
TEST('ExitingFiresOneShotAfterPermsAutoSatisfied');

// With no mapped perms, FB_Permissives' unmapped-bits-are-good policy
// means bOK is TRUE from scan one. After Entry (scan 1) and the
// settle-Execute (scan 2), scan 3 must surface Exiting as a one-shot
// cleanup hook before the Advance phase takes over.
Setup();
sm.SetCurrentStep(nStep := 3000);

step(sm := sm, nStep := 3000, nNextStep := 3002, nTimeout := 0, sName := 'Exit');
step(sm := sm, nStep := 3000, nNextStep := 3002, nTimeout := 0, sName := 'Exit');
step(sm := sm, nStep := 3000, nNextStep := 3002, nTimeout := 0, sName := 'Exit');

AssertFalse(
    Condition := step.Entry,
    Message   := 'Entry must stay FALSE on the Exiting scan');
AssertFalse(
    Condition := step.Execute,
    Message   := 'Execute must drop once perms are satisfied, so Exiting can run');
AssertTrue(
    Condition := step.Exiting,
    Message   := 'Exiting must pulse TRUE once after perms go satisfied');

TEST_FINISHED();
END_METHOD

METHOD AdvancePhaseKeepsAllLifecycleOutputsClear
VAR
    step : TcForge.FB_Step;
END_VAR
TEST('AdvancePhaseKeepsAllLifecycleOutputsClear');

// After Entry, settle-Execute and Exiting have fired, FB_Step is in the
// Advance branch, which calls sm.SetNextStep every scan and leaves all
// three lifecycle outputs FALSE. Confirms Exiting is a true one-shot
// (not sticky) and user code won't see stale Exit work on later scans.
Setup();
sm.SetCurrentStep(nStep := 3000);

step(sm := sm, nStep := 3000, nNextStep := 3002, nTimeout := 0, sName := 'Adv');
step(sm := sm, nStep := 3000, nNextStep := 3002, nTimeout := 0, sName := 'Adv');
step(sm := sm, nStep := 3000, nNextStep := 3002, nTimeout := 0, sName := 'Adv');
step(sm := sm, nStep := 3000, nNextStep := 3002, nTimeout := 0, sName := 'Adv');

AssertFalse(
    Condition := step.Entry,
    Message   := 'Entry must stay FALSE in the Advance phase');
AssertFalse(
    Condition := step.Execute,
    Message   := 'Execute must stay FALSE in the Advance phase');
AssertFalse(
    Condition := step.Exiting,
    Message   := 'Exiting must stay FALSE in the Advance phase (one-shot, not sticky)');

TEST_FINISHED();
END_METHOD

METHOD NamePublishedIntoSmStepInfo
VAR
    step : TcForge.FB_Step;
END_VAR
TEST('NamePublishedIntoSmStepInfo');

// While a step is active it must publish its human-readable name into
// sm.Status.Step.Name so HMI / diagnostics can show what is currently
// running. The name comes straight from the sName VAR_INPUT each scan.
Setup();
sm.SetCurrentStep(nStep := 3000);

step(sm := sm, nStep := 3000, nNextStep := 3002, nTimeout := 0,
     sName := 'Advance cylinder');

AssertEquals_STRING(
    Expected := 'Advance cylinder',
    Actual   := sm.Status.Step.Name,
    Message  := 'Active step must publish its sName into sm.Status.Step.Name');

TEST_FINISHED();
END_METHOD

METHOD MappedFalsePermHoldsExecuteAndBlocksExit
VAR
    step : TcForge.FB_Step;
    i    : INT;
END_VAR
TEST('MappedFalsePermHoldsExecuteAndBlocksExit');

// A mapped permissive that is not satisfied must keep Execute firing
// every scan while the step waits, and must never let Exiting fire.
// The step is stuck in the "waiting for perms" Execute branch.
Setup();
sm.SetCurrentStep(nStep := 3000);

FOR i := 1 TO 6 DO
    step.MapPerm(nIndex := 0, sDescription := 'Sensor A', bValue := FALSE);
    step(sm := sm, nStep := 3000, nNextStep := 3002,
         nTimeout := 0, sName := 'WaitingPerm');
END_FOR;

AssertFalse(
    Condition := step.Entry,
    Message   := 'Entry must be FALSE while the step is waiting on a failing perm');
AssertTrue(
    Condition := step.Execute,
    Message   := 'Execute must keep firing every scan while perms are unsatisfied');
AssertFalse(
    Condition := step.Exiting,
    Message   := 'Exiting must not fire while any mapped perm is still FALSE');

TEST_FINISHED();
END_METHOD

METHOD MappedTruePermLetsExitFireAfterSettle
VAR
    step : TcForge.FB_Step;
    i    : INT;
    sawExiting : BOOL;
END_VAR
TEST('MappedTruePermLetsExitFireAfterSettle');

// Hold a mapped permissive FALSE for a few scans (Execute stays high),
// then flip it TRUE. After the perm-settle pass Exiting must fire
// exactly once as a one-shot on its way into Advance. We loop a few
// scans after the flip and latch whether Exiting was ever observed.
Setup();
sm.SetCurrentStep(nStep := 3000);

FOR i := 1 TO 3 DO
    step.MapPerm(nIndex := 0, sDescription := 'Sensor A', bValue := FALSE);
    step(sm := sm, nStep := 3000, nNextStep := 3002,
         nTimeout := 0, sName := 'WaitThenPass');
END_FOR;

sawExiting := FALSE;
FOR i := 1 TO 4 DO
    step.MapPerm(nIndex := 0, sDescription := 'Sensor A', bValue := TRUE);
    step(sm := sm, nStep := 3000, nNextStep := 3002,
         nTimeout := 0, sName := 'WaitThenPass');
    IF step.Exiting THEN
        sawExiting := TRUE;
    END_IF;
END_FOR;

AssertTrue(
    Condition := sawExiting,
    Message   := 'Exiting must fire on the scan after the mapped perm flips to TRUE');

TEST_FINISHED();
END_METHOD

METHOD ZeroTimeoutNeverRaisesTimeoutFault
VAR
    step : TcForge.FB_Step;
    i    : INT;
END_VAR
TEST('ZeroTimeoutNeverRaisesTimeoutFault');

// nTimeout = 0 is the "disabled" convention: the timeout branch must
// not fire regardless of TimerSeconds. We inject a large TimerSeconds
// directly via the probe so we do not need to actually let time pass,
// and we hold a perm FALSE so we stay in the Execute-wait branch
// (which is where the timeout check lives).
Setup();
sm.SetCurrentStep(nStep := 3000);
sm.SetTimerSeconds(seconds := 99999.0);

FOR i := 1 TO 5 DO
    step.MapPerm(nIndex := 0, sDescription := 'Sensor A', bValue := FALSE);
    step(sm := sm, nStep := 3000, nNextStep := 3002,
         nTimeout := 0, sName := 'NoTimeout');
END_FOR;

AssertEquals_DINT(
    Expected := 0,
    Actual   := sm.GetFaultCode(),
    Message  := 'nTimeout = 0 must keep the timeout branch disabled, no fault raised');

TEST_FINISHED();
END_METHOD

METHOD TimeoutRaisesStepTimeoutFault
VAR
    step : TcForge.FB_Step;
    i    : INT;
END_VAR
TEST('TimeoutRaisesStepTimeoutFault');

// With TimerSeconds past nTimeout and perms not satisfied, FB_Step
// must route a StepTimeout fault through sm._RaiseStepFault so the
// inherited ring buffer picks it up. We observe the result via
// sm.GetFaultCode() (inherited diagnostics from FB_DeviceBase).
Setup();
sm.SetCurrentStep(nStep := 3000);
sm.SetTimerSeconds(seconds := 12.0);

FOR i := 1 TO 4 DO
    step.MapPerm(nIndex := 0, sDescription := 'Sensor A', bValue := FALSE);
    step(sm := sm, nStep := 3000, nNextStep := 3002,
         nTimeout := 5, sName := 'WillTimeout');
END_FOR;

AssertEquals_DINT(
    Expected := TcForge.E_SM_Fault.StepTimeout,
    Actual   := sm.GetFaultCode(),
    Message  := 'Expired step timeout must raise E_SM_Fault.StepTimeout on the SM');

TEST_FINISHED();
END_METHOD

METHOD InactiveRaiseFaultIsNoOp
VAR
    step : TcForge.FB_Step;
END_VAR
TEST('InactiveRaiseFaultIsNoOp');

// RaiseFault is documented as "only legal inside a step block"; the FB
// must early-return when _active is FALSE so a stray call from the
// wrong scope does not corrupt the SM fault state.
Setup();

step(sm := sm, nStep := 3000, nNextStep := 3002, nTimeout := 0, sName := 'Idle');
step.RaiseFault(code := TcForge.E_SM_Fault.StepUserFault, reason := 'Should not land');

AssertEquals_DINT(
    Expected := 0,
    Actual   := sm.GetFaultCode(),
    Message  := 'RaiseFault on an inactive step must be a no-op');

TEST_FINISHED();
END_METHOD

METHOD RaiseFaultWhileActiveRecordsCode
VAR
    step : TcForge.FB_Step;
END_VAR
TEST('RaiseFaultWhileActiveRecordsCode');

// When called while the step is active, RaiseFault must push the code
// and reason through sm._RaiseStepFault so the SM's fault handling
// records it. The companion SetNextStep(nStep + 1) jump is exercised
// end-to-end by the FB_StateMachine suite; here we only lock in the
// fault-recording contract that FB_DeviceBase exposes via GetFaultCode.
Setup();
sm.SetCurrentStep(nStep := 3000);

step(sm := sm, nStep := 3000, nNextStep := 3002, nTimeout := 0, sName := 'UserFault');
step.RaiseFault(
    code   := TcForge.E_SM_Fault.StepUserFault,
    reason := 'Sensor A out of range');

AssertEquals_DINT(
    Expected := TcForge.E_SM_Fault.StepUserFault,
    Actual   := sm.GetFaultCode(),
    Message  := 'Active-step RaiseFault must surface its code through sm.GetFaultCode');

TEST_FINISHED();
END_METHOD

END_FUNCTION_BLOCK

// ---- POUs/FB_StateMachine_Probe.TcPOU
// Test-only child of FB_StateMachine. Two jobs:
//
//   1. Shift internals (state, step, timer, _nextStep, permissives) into
//      test reach. FB_StateMachine publishes Status as VAR_OUTPUT (which
//      TwinCAT makes read-only from outside) and keeps its permission /
//      interlock blocks as plain VAR members with no external mapping
//      API, so tests cannot drive them without a subclass.
//
//   2. Drive the parent body when the test wants it (SUPER^()) and skip
//      it when the test doesn't. FB_Step_Test never calls sm() on the
//      probe — it only uses the mutators and the step FB under test
//      drives its own observables. FB_StateMachine_Test does call sm()
//      to exercise transitions. Because the body is just SUPER^(),
//      both uses are safe: invoking sm() runs the parent logic,
//      skipping it leaves the injected test state put.
//
// Access note: FB_StateMachine declares permAuto / permHome / permStart
// / permProceed / intlkRunning / R_TRIG_1 / R_TRIG_5 / _nextStep and
// the _*Requested command flags as plain `VAR`, which in TwinCAT is
// accessible to subclasses (PROTECTED-like default). This probe leans
// on that — none of these mutators compile if the parent hides them.
//
// Lives in the Testing project only — not part of TcForge's public API.
FUNCTION_BLOCK FB_StateMachine_Probe EXTENDS TcForge.FB_StateMachine

SUPER^();

// Full isolation reset for the shared suite-level probe. Clears fault
// book-keeping, command-request flags, permissive / interlock live
// state, rising-edge memory on the SM's internal triggers, and
// published Status back to its power-on values. Each test method
// calls this in its own Setup() so tests see a clean slate even
// though the probe instance itself is reused.
//
// Why rising edges matter: R_TRIG_5 fires _completeStateRequested
// when the current step is in-range for the state AND _nextStep=0.
// In STOPPED with Step.Current=0 that condition is trivially TRUE
// (STOPPED has no step range, _IsStepInStateRange returns a
// degenerate [0,0] match), so a fresh probe or a previous test
// leaves the rising-edge memory armed — we must explicitly drive
// CLK:=FALSE to clear it.
METHOD PUBLIC ResetAll
VAR
    rsp : TcForge.E_RpcMethodResponse;
END_VAR
rsp := Reset();

_abortRequested         := FALSE;
_completeStateRequested := FALSE;
_homeRequested          := FALSE;
_pauseRequested         := FALSE;
_proceedRequested       := FALSE;
_startRequested         := FALSE;
_stopRequested          := FALSE;
_retryActive            := FALSE;
RetryComplete           := FALSE;
_blockedCode            := 0;
_starvedCode            := 0;

// Order matters for FB_Interlock: Reset() snaps _latchedBits to the
// current nLiveBits, so the live bits must already be good before the
// reset. Otherwise a bit left FALSE by a previous test (e.g. the
// running-interlock-trip case) stays latched bad across the reset and
// makes every subsequent test look like the interlock auto-aborted.
// FB_Permissives is non-latching so the order doesn't matter there,
// but we keep it consistent.
permHome.MapInput(bitIndex := 0, inputValue := TRUE);
permStart.MapInput(bitIndex := 0, inputValue := TRUE);
permProceed.MapInput(bitIndex := 0, inputValue := TRUE);
permAuto.MapInput(bitIndex := 0, inputValue := TRUE);
intlkRunning.MapInput(bitIndex := 0, inputValue := TRUE);
permHome.Reset();
permStart.Reset();
permProceed.Reset();
permAuto.Reset();
intlkRunning.Reset();

R_TRIG_1(CLK := FALSE);
R_TRIG_5(CLK := FALSE);

Status.State            := TcForge.E_SM_State.STOPPED;
Status.LastState        := TcForge.E_SM_State.STOPPED;
Status.Step.Current     := 0;
Status.Step.Next        := 0;
Status.Step.TimerSeconds := 0.0;
Status.Faulted          := FALSE;
Status.SubmoduleFaulted := FALSE;
Status.BlockedCondition := 0;
Status.StarvedCondition := 0;
Status.AutoStartRequest := FALSE;
Status.AutoCycleRequest := FALSE;

_nextStep      := 0;
_returnState   := TcForge.E_SM_State.STOPPED;
ReturnNextStep := 0;
PreviousStep   := 0;
END_METHOD

// Force the active step number. Lets FB_Step see _active = TRUE without
// us having to drive Home/Start/state transitions end-to-end.
METHOD PUBLIC SetCurrentStep
VAR_INPUT
    nStep : DINT;
END_VAR
Status.Step.Current := nStep;
END_METHOD

// Inject a step-timer reading so timeout branches can be tested without
// actually letting wall-clock time pass. The production SM owns the
// timer — here we just write the published value directly.
METHOD PUBLIC SetTimerSeconds
VAR_INPUT
    seconds : REAL;
END_VAR
Status.Step.TimerSeconds := seconds;
END_METHOD

// Park the SM in a specific state without walking the full
// Home/Start/Complete command sequence. Used by the transition tests
// to set up "machine is in state X, now issue command Y" without
// running a sequence first.
METHOD PUBLIC ForceState
VAR_INPUT
    state : TcForge.E_SM_State;
END_VAR
Status.State := state;
END_METHOD

// Set Status.LastState directly. Needed for the AutoCycle path
// (fires when State=READY AND LastState=RUNNING) without walking
// a full RUNNING -> READY transition first.
METHOD PUBLIC ForceLastState
VAR_INPUT
    state : TcForge.E_SM_State;
END_VAR
Status.LastState := state;
END_METHOD

// Drive _nextStep directly. Used with ForceState+SetCurrentStep to
// simulate "mid-sequence" — if _nextStep stays at 0 while a forced
// Current lands inside the state's step range, R_TRIG_5 fires a
// spurious sequence-complete that tests don't want.
METHOD PUBLIC ForceNextStep
VAR_INPUT
    nStep : DINT;
END_VAR
_nextStep := nStep;
END_METHOD

// Map a bit into the private permHome block so the Home-permissive
// gate can be observed. Without this the internal FB_Permissives has
// no external mapping surface on the SM, and every test would see
// "all perms OK" by default.
METHOD PUBLIC MapHomePerm
VAR_INPUT
    bitIndex : UDINT;
    bGood    : BOOL;
END_VAR
permHome.MapInput(bitIndex := bitIndex, inputValue := bGood);
END_METHOD

METHOD PUBLIC MapStartPerm
VAR_INPUT
    bitIndex : UDINT;
    bGood    : BOOL;
END_VAR
permStart.MapInput(bitIndex := bitIndex, inputValue := bGood);
END_METHOD

METHOD PUBLIC MapProceedPerm
VAR_INPUT
    bitIndex : UDINT;
    bGood    : BOOL;
END_VAR
permProceed.MapInput(bitIndex := bitIndex, inputValue := bGood);
END_METHOD

METHOD PUBLIC MapAutoPerm
VAR_INPUT
    bitIndex : UDINT;
    bGood    : BOOL;
END_VAR
permAuto.MapInput(bitIndex := bitIndex, inputValue := bGood);
END_METHOD

END_FUNCTION_BLOCK

// ---- Tests/FB_StateMachine_Test.TcPOU
// Tests for FB_StateMachine, the sequencing core: command gating,
// state transitions, permissive enforcement, running interlock,
// fault surfacing, and OEE condition reporting. We drive the SM
// through its public command API (Home/Start/Stop/Pause/Proceed/
// Abort/ReportBlocked/ReportStarved) and observe Status.
//
// Test strategy: FB_StateMachine_Probe runs SUPER^() in its body,
// so calling sm() exercises the real parent logic. The probe also
// exposes ResetAll / ForceState / ForceLastState / SetCurrentStep /
// ForceNextStep / Map*Perm to park the SM in an arbitrary state
// without walking a full sequence first — otherwise every test
// would have to start from STOPPED and drive Home -> HOMING ->
// READY before it could observe a RUNNING-state transition.
//
// Shared-sm note: FB_StateMachine is ~52 KB and TwinCAT puts
// method-local VAR on the task stack (default 48 KB), so a probe
// per test overflows the stack (C0297) and takes the runtime down
// at activation. The probe is therefore declared at the suite FB
// level and each test calls sm.ResetAll() at the top to clear
// state / faults / triggers between tests. See FB_Step_Test for
// the first time we hit this and the resolution write-up.
FUNCTION_BLOCK FB_StateMachine_Test EXTENDS TcUnit.FB_TestSuite
VAR
    sm : FB_StateMachine_Probe;
END_VAR

FreshSmIsStoppedAtStepZero();
HomeFromStoppedEntersHomingAtMinStep();
HomeFromRunningRejectedWrongState();
HomeRejectedWhenHomePermBad();
StartFromReadyEntersRunningAtMinStep();
StartRejectedFromStopped();
StopFromRunningEntersStopping();
StopFromReadyGoesStraightToStopped();
AbortFromRunningEntersAborting();
AbortRejectedFromStopped();
PauseFromRunningEntersPausing();
ProceedFromPausedEntersProceeding();
HomingCompletesToReadyOnNextStepZero();
RunningInterlockTripAutoAbortsWithFault();
OddStepCurrentAutoRaisesOddStepReached();
SubmoduleFaultInputRaisesSubmoduleFaulted();
BlockedConditionPublishedDuringRunning();

METHOD FreshSmIsStoppedAtStepZero
TEST('FreshSmIsStoppedAtStepZero');

// Baseline: power-on defaults. WaitingState TRUE, ActiveState FALSE,
// Faulted FALSE, no fault code, Step.Current=0. This also verifies that
// ResetAll puts the shared probe back to the first-boot contract between
// tests instead of carrying over state from the previous case.
sm.ResetAll();
sm();

AssertEquals_DINT(
    Expected := TcForge.E_SM_State.STOPPED,
    Actual   := sm.Status.State,
    Message  := 'Fresh SM must report State = STOPPED');
AssertEquals_DINT(
    Expected := DINT#0,
    Actual   := sm.Status.Step.Current,
    Message  := 'Fresh SM must report Step.Current = 0');
AssertTrue(
    Condition := sm.Status.WaitingState,
    Message   := 'Fresh SM must report WaitingState = TRUE');
AssertFalse(
    Condition := sm.Status.ActiveState,
    Message   := 'Fresh SM must not report ActiveState');
AssertEquals_DINT(
    Expected := DINT#0,
    Actual   := sm.GetFaultCode(),
    Message  := 'Fresh SM must report no fault');

TEST_FINISHED();
END_METHOD

METHOD HomeFromStoppedEntersHomingAtMinStep
VAR
    rsp : TcForge.E_RpcMethodResponse;
END_VAR
TEST('HomeFromStoppedEntersHomingAtMinStep');

// Stopped + Home -> Homing, auto-init to HOMING_MIN (1000). Validates the
// happy-path command gate (Home only accepted in STOPPED) and the
// auto-init-first-step-on-entering-active-state behaviour in one pass.
sm.ResetAll();

rsp := sm.Home();
AssertEquals_DINT(
    Expected := TcForge.E_RpcMethodResponse.ACCEPTED,
    Actual   := rsp,
    Message  := 'Home() must be ACCEPTED from STOPPED with perms OK');

sm();

AssertEquals_DINT(
    Expected := TcForge.E_SM_State.HOMING,
    Actual   := sm.Status.State,
    Message  := 'Home from STOPPED must transition State to HOMING');
AssertEquals_DINT(
    Expected := DINT#1000,
    Actual   := sm.Status.Step.Current,
    Message  := 'Entering HOMING must auto-init Step.Current to HOMING_MIN (1000)');
AssertTrue(
    Condition := sm.Status.ActiveState,
    Message   := 'HOMING must report ActiveState = TRUE');

TEST_FINISHED();
END_METHOD

METHOD HomeFromRunningRejectedWrongState
VAR
    rsp : TcForge.E_RpcMethodResponse;
END_VAR
TEST('HomeFromRunningRejectedWrongState');

// Home is only valid from STOPPED. From RUNNING it must be rejected with
// REJECTED_WRONG_STATE and must not set the internal _homeRequested flag,
// so a subsequent sm() does not transition.
sm.ResetAll();
sm.ForceState(state := TcForge.E_SM_State.RUNNING);
sm.SetCurrentStep(nStep := 3000);
sm.ForceNextStep(nStep := 3002);

rsp := sm.Home();
AssertEquals_DINT(
    Expected := TcForge.E_RpcMethodResponse.REJECTED_WRONG_STATE,
    Actual   := rsp,
    Message  := 'Home() from RUNNING must return REJECTED_WRONG_STATE');

sm();

AssertEquals_DINT(
    Expected := TcForge.E_SM_State.RUNNING,
    Actual   := sm.Status.State,
    Message  := 'State must stay RUNNING when Home() is rejected');

TEST_FINISHED();
END_METHOD

METHOD HomeRejectedWhenHomePermBad
VAR
    rsp : TcForge.E_RpcMethodResponse;
END_VAR
TEST('HomeRejectedWhenHomePermBad');

// Permissive gate: Home must be rejected with REJECTED_PERMISSIVE_NOT_MET
// when permHome.sts.bOK is FALSE. We need one body scan after mapping
// the bad bit so permHome() recomputes sts.bOK before Home() reads it.
sm.ResetAll();
sm.MapHomePerm(bitIndex := 1, bGood := FALSE);
sm();

rsp := sm.Home();
AssertEquals_DINT(
    Expected := TcForge.E_RpcMethodResponse.REJECTED_PERMISSIVE_NOT_MET,
    Actual   := rsp,
    Message  := 'Home() with permHome bad must return REJECTED_PERMISSIVE_NOT_MET');

AssertEquals_DINT(
    Expected := TcForge.E_SM_State.STOPPED,
    Actual   := sm.Status.State,
    Message  := 'State must stay STOPPED when Home() is rejected on perms');

TEST_FINISHED();
END_METHOD

METHOD StartFromReadyEntersRunningAtMinStep
VAR
    rsp : TcForge.E_RpcMethodResponse;
END_VAR
TEST('StartFromReadyEntersRunningAtMinStep');

// Ready + Start -> Running, auto-init to RUNNING_MIN (3000). Parks the
// SM directly in READY since the Home -> Homing -> Ready walk would
// require a full step sequence and is covered elsewhere.
sm.ResetAll();
sm.ForceState(state := TcForge.E_SM_State.READY);

rsp := sm.Start();
AssertEquals_DINT(
    Expected := TcForge.E_RpcMethodResponse.ACCEPTED,
    Actual   := rsp,
    Message  := 'Start() must be ACCEPTED from READY with perms OK');

sm();

AssertEquals_DINT(
    Expected := TcForge.E_SM_State.RUNNING,
    Actual   := sm.Status.State,
    Message  := 'Start from READY must transition State to RUNNING');
AssertEquals_DINT(
    Expected := DINT#3000,
    Actual   := sm.Status.Step.Current,
    Message  := 'Entering RUNNING must auto-init Step.Current to RUNNING_MIN (3000)');

TEST_FINISHED();
END_METHOD

METHOD StartRejectedFromStopped
VAR
    rsp : TcForge.E_RpcMethodResponse;
END_VAR
TEST('StartRejectedFromStopped');

// Start only valid from READY — STOPPED must reject with WRONG_STATE so
// users cannot skip homing. A rejected Start must not leave the machine
// queued for an auto-start on the next cycle.
sm.ResetAll();

rsp := sm.Start();
AssertEquals_DINT(
    Expected := TcForge.E_RpcMethodResponse.REJECTED_WRONG_STATE,
    Actual   := rsp,
    Message  := 'Start() from STOPPED must return REJECTED_WRONG_STATE');

sm();

AssertEquals_DINT(
    Expected := TcForge.E_SM_State.STOPPED,
    Actual   := sm.Status.State,
    Message  := 'State must stay STOPPED when Start() is rejected');

TEST_FINISHED();
END_METHOD

METHOD StopFromRunningEntersStopping
VAR
    rsp : TcForge.E_RpcMethodResponse;
END_VAR
TEST('StopFromRunningEntersStopping');

// Running + Stop -> Stopping: the graceful shutdown path. ForceNextStep
// keeps us mid-sequence so R_TRIG_5 does not pre-fire a spurious
// sequence-complete on this scan.
sm.ResetAll();
sm.ForceState(state := TcForge.E_SM_State.RUNNING);
sm.SetCurrentStep(nStep := 3000);
sm.ForceNextStep(nStep := 3002);

rsp := sm.Stop();
AssertEquals_DINT(
    Expected := TcForge.E_RpcMethodResponse.ACCEPTED,
    Actual   := rsp,
    Message  := 'Stop() must be ACCEPTED from RUNNING');

sm();

AssertEquals_DINT(
    Expected := TcForge.E_SM_State.STOPPING,
    Actual   := sm.Status.State,
    Message  := 'Stop from RUNNING must transition State to STOPPING');

TEST_FINISHED();
END_METHOD

METHOD StopFromReadyGoesStraightToStopped
VAR
    rsp : TcForge.E_RpcMethodResponse;
END_VAR
TEST('StopFromReadyGoesStraightToStopped');

// Ready is already quiescent (no sequence to shut down), so Stop skips
// Stopping entirely and lands in STOPPED on the same scan. This avoids
// the HMI lie of "stopping" when there is nothing to stop.
sm.ResetAll();
sm.ForceState(state := TcForge.E_SM_State.READY);

rsp := sm.Stop();
AssertEquals_DINT(
    Expected := TcForge.E_RpcMethodResponse.ACCEPTED,
    Actual   := rsp,
    Message  := 'Stop() must be ACCEPTED from READY');

sm();

AssertEquals_DINT(
    Expected := TcForge.E_SM_State.STOPPED,
    Actual   := sm.Status.State,
    Message  := 'Stop from READY must transition directly to STOPPED');

TEST_FINISHED();
END_METHOD

METHOD AbortFromRunningEntersAborting
VAR
    rsp : TcForge.E_RpcMethodResponse;
END_VAR
TEST('AbortFromRunningEntersAborting');

// Abort is accepted from any state except STOPPED / ABORTING. From
// RUNNING it transitions to ABORTING on the first body scan with
// Step.Current reset to 0 (the transition sets _nextStep:=0 and
// step-mgmt propagates it). Auto-init to ABORTING_MIN (5000) happens
// on the NEXT scan when R_TRIG_1 fires on Current=0 and the
// "enter-active-state" branch picks the new min. Two scans is the
// real SM contract — tested explicitly here because it trips up
// any consumer expecting a one-scan settle.
sm.ResetAll();
sm.ForceState(state := TcForge.E_SM_State.RUNNING);
sm.SetCurrentStep(nStep := 3000);
sm.ForceNextStep(nStep := 3002);

rsp := sm.Abort();
AssertEquals_DINT(
    Expected := TcForge.E_RpcMethodResponse.ACCEPTED,
    Actual   := rsp,
    Message  := 'Abort() must be ACCEPTED from RUNNING');

sm();
AssertEquals_DINT(
    Expected := TcForge.E_SM_State.ABORTING,
    Actual   := sm.Status.State,
    Message  := 'Abort from RUNNING must transition State to ABORTING on first scan');
AssertEquals_DINT(
    Expected := DINT#0,
    Actual   := sm.Status.Step.Current,
    Message  := 'Abort from RUNNING must reset Step.Current to 0 on the transition scan');

sm();
AssertEquals_DINT(
    Expected := DINT#5000,
    Actual   := sm.Status.Step.Current,
    Message  := 'Second scan after entering ABORTING must auto-init Step.Current to ABORTING_MIN (5000)');

TEST_FINISHED();
END_METHOD

METHOD AbortRejectedFromStopped
VAR
    rsp : TcForge.E_RpcMethodResponse;
END_VAR
TEST('AbortRejectedFromStopped');

// Already-stopped machine: Abort is a no-op and must report
// REJECTED_WRONG_STATE rather than silently staying accepted.
// Prevents the HMI from thinking it just triggered a new abort episode.
sm.ResetAll();

rsp := sm.Abort();
AssertEquals_DINT(
    Expected := TcForge.E_RpcMethodResponse.REJECTED_WRONG_STATE,
    Actual   := rsp,
    Message  := 'Abort() from STOPPED must return REJECTED_WRONG_STATE');

TEST_FINISHED();
END_METHOD

METHOD PauseFromRunningEntersPausing
VAR
    rsp : TcForge.E_RpcMethodResponse;
END_VAR
TEST('PauseFromRunningEntersPausing');

// Running + Pause -> Pausing, and the SM must remember the step we were
// on (ReturnNextStep) so Proceed can resume at the same spot. We only
// assert state here; the save/restore round-trip is covered by
// ProceedFromPausedEntersProceeding.
sm.ResetAll();
sm.ForceState(state := TcForge.E_SM_State.RUNNING);
sm.SetCurrentStep(nStep := 3000);
sm.ForceNextStep(nStep := 3002);

rsp := sm.Pause();
AssertEquals_DINT(
    Expected := TcForge.E_RpcMethodResponse.ACCEPTED,
    Actual   := rsp,
    Message  := 'Pause() must be ACCEPTED from RUNNING');

sm();

AssertEquals_DINT(
    Expected := TcForge.E_SM_State.PAUSING,
    Actual   := sm.Status.State,
    Message  := 'Pause from RUNNING must transition State to PAUSING');

TEST_FINISHED();
END_METHOD

METHOD ProceedFromPausedEntersProceeding
VAR
    rsp : TcForge.E_RpcMethodResponse;
END_VAR
TEST('ProceedFromPausedEntersProceeding');

// Paused + Proceed -> Proceeding: the sequence-resume path. Only valid
// from PAUSED; the transition relies on permProceed and permAuto both
// OK, which ResetAll leaves TRUE by default.
sm.ResetAll();
sm.ForceState(state := TcForge.E_SM_State.PAUSED);

rsp := sm.Proceed();
AssertEquals_DINT(
    Expected := TcForge.E_RpcMethodResponse.ACCEPTED,
    Actual   := rsp,
    Message  := 'Proceed() must be ACCEPTED from PAUSED');

sm();

AssertEquals_DINT(
    Expected := TcForge.E_SM_State.PROCEEDING,
    Actual   := sm.Status.State,
    Message  := 'Proceed from PAUSED must transition State to PROCEEDING');

TEST_FINISHED();
END_METHOD

METHOD HomingCompletesToReadyOnNextStepZero
TEST('HomingCompletesToReadyOnNextStepZero');

// Sequence completion inference: the SM treats "current step is in the
// HOMING range AND _nextStep = 0" as "the last step just finished".
// R_TRIG_5 fires, _completeStateRequested latches, the Homing-complete
// transition fires in the same scan, State becomes READY, and LastState
// gets HOMING so auto-cycle book-keeping can tell what just ran.
sm.ResetAll();
sm.ForceState(state := TcForge.E_SM_State.HOMING);
sm.SetCurrentStep(nStep := 1005);
sm.ForceNextStep(nStep := 0);

sm();

AssertEquals_DINT(
    Expected := TcForge.E_SM_State.READY,
    Actual   := sm.Status.State,
    Message  := 'HOMING with _nextStep=0 at in-range step must complete to READY');
AssertEquals_DINT(
    Expected := TcForge.E_SM_State.HOMING,
    Actual   := sm.Status.LastState,
    Message  := 'After HOMING->READY, LastState must be HOMING');

TEST_FINISHED();
END_METHOD

METHOD RunningInterlockTripAutoAbortsWithFault
TEST('RunningInterlockTripAutoAbortsWithFault');

// intlkRunning trip from any active state must auto-abort and raise
// RunningInterlockTripped through the shared fault book-keeping. The
// state goes to ABORTING on the same scan the interlock body sees the
// bad bit, no additional command needed.
sm.ResetAll();
sm.ForceState(state := TcForge.E_SM_State.RUNNING);
sm.SetCurrentStep(nStep := 3000);
sm.ForceNextStep(nStep := 3002);
sm.MapRunningIntlk(bitIndex := 0, bGood := FALSE);

sm();

AssertEquals_DINT(
    Expected := TcForge.E_SM_State.ABORTING,
    Actual   := sm.Status.State,
    Message  := 'Running interlock trip from RUNNING must auto-transition to ABORTING');
AssertEquals_DINT(
    Expected := TcForge.E_SM_Fault.RunningInterlockTripped,
    Actual   := sm.GetFaultCode(),
    Message  := 'Running interlock trip must raise RunningInterlockTripped');

TEST_FINISHED();
END_METHOD

METHOD OddStepCurrentAutoRaisesOddStepReached
TEST('OddStepCurrentAutoRaisesOddStepReached');

// Convention: odd step numbers are fault landing pads. When Step.Current
// is odd and no more specific fault has been raised yet, the SM body
// publishes Status.Faulted=TRUE and raises the default OddStepReached
// code. A specific raise (StepTimeout, StepUserFault, submodule, ...)
// that fired earlier would win thanks to the GetFaultCode()=0 guard.
//
// _nextStep must stay pinned to the same odd step — if we let it be a
// neighbour, step-mgmt advances Current off the odd value before the
// fault check runs and LsOdd comes out 0.
sm.ResetAll();
sm.ForceState(state := TcForge.E_SM_State.RUNNING);
sm.SetCurrentStep(nStep := 3001);
sm.ForceNextStep(nStep := 3001);

sm();

AssertTrue(
    Condition := sm.Status.Faulted,
    Message   := 'Odd Step.Current must set Status.Faulted = TRUE');
AssertEquals_DINT(
    Expected := TcForge.E_SM_Fault.OddStepReached,
    Actual   := sm.GetFaultCode(),
    Message  := 'Odd Step.Current must raise default OddStepReached when no other fault active');

TEST_FINISHED();
END_METHOD

METHOD SubmoduleFaultInputRaisesSubmoduleFaulted
TEST('SubmoduleFaultInputRaisesSubmoduleFaulted');

// External submodule fault hook: inpSubmoduleFaulted=TRUE must publish
// Status.SubmoduleFaulted and raise the SubmoduleFaulted fault code so
// parent supervisors see a matching ST_DeviceHeader_Sts entry. We park
// in STOPPED with an even step so OddStepReached doesn't race ahead.
sm.ResetAll();
sm.inpSubmoduleFaulted := TRUE;

sm();

AssertTrue(
    Condition := sm.Status.SubmoduleFaulted,
    Message   := 'inpSubmoduleFaulted must surface on Status.SubmoduleFaulted');
AssertEquals_DINT(
    Expected := TcForge.E_SM_Fault.SubmoduleFaulted,
    Actual   := sm.GetFaultCode(),
    Message  := 'inpSubmoduleFaulted must raise SubmoduleFaulted through fault book-keeping');

sm.inpSubmoduleFaulted := FALSE;

TEST_FINISHED();
END_METHOD

METHOD BlockedConditionPublishedDuringRunning
TEST('BlockedConditionPublishedDuringRunning');

// OEE reporting: ReportBlocked(code) stashes an internal latch that the
// body consumes once per cycle when the SM is in a producing state
// (RUNNING / STOPPING / READY) and publishes on Status.BlockedCondition.
// Calling from STOPPED alone would not publish — the guard is what
// prevents stale condition codes from looking like active blockage.
sm.ResetAll();
sm.ForceState(state := TcForge.E_SM_State.RUNNING);
sm.SetCurrentStep(nStep := 3000);
sm.ForceNextStep(nStep := 3002);

sm.ReportBlocked(code := DINT#42);
sm();

AssertEquals_DINT(
    Expected := DINT#42,
    Actual   := sm.Status.BlockedCondition,
    Message  := 'ReportBlocked(42) during RUNNING must publish Status.BlockedCondition = 42');

TEST_FINISHED();
END_METHOD

END_FUNCTION_BLOCK

// ---- POUs/FB_DigitalInput_Probe.TcPOU
// Test-only child of FB_DigitalInput. The production FB keeps `io` in its
// private VAR section so external callers can't poke the hardware-linked
// struct; this probe adds a SetRawInput() method so FB_DigitalInput_Test
// can inject the raw wire value each cycle without touching the public
// surface.
//
// Lives in the Testing project only — not part of TcForge's public API.
FUNCTION_BLOCK FB_DigitalInput_Probe EXTENDS TcForge.FB_DigitalInput

// Delegate the cyclic body to FB_DigitalInput. In IEC 61131-3 the child's
// implementation REPLACES the parent's; SUPER^() is required to run the
// inherited conditioning pipeline against the probe's injected value.
SUPER^();

// Drive the internal hardware-linked bit. Call immediately before the
// cyclic body runs to simulate a physical transition.
METHOD PUBLIC SetRawInput
VAR_INPUT
    bValue : BOOL;
END_VAR
io.inSignal := bValue;
END_METHOD

END_FUNCTION_BLOCK

// ---- POUs/FB_TwoPosActuator_Probe.TcPOU
// Test-only child of FB_TwoPosActuator. The production FB keeps io,
// advancePermissives, and retractPermissives in its private VAR section,
// so tests use this probe to inject field signals and map permissives
// without touching the public surface.
//
// The probe delegates the cyclic body back to the parent via SUPER^() —
// without that call the child's empty body would replace the parent's
// state-machine logic and every assertion would see zeroed state.
//
// Lives in the Testing project only — not part of TcForge's public API.
FUNCTION_BLOCK FB_TwoPosActuator_Probe EXTENDS TcForge.FB_TwoPosActuator

// Run the inherited state machine using the probe's injected signals.
SUPER^();

METHOD PUBLIC SetAdvancedFeedback
VAR_INPUT
    bValue : BOOL;
END_VAR
io.inFbkAdvanced := bValue;
END_METHOD

METHOD PUBLIC SetRetractedFeedback
VAR_INPUT
    bValue : BOOL;
END_VAR
io.inFbkRetracted := bValue;
END_METHOD

METHOD PUBLIC GetValveAdvance : BOOL
GetValveAdvance := io.outValveAdvance;
END_METHOD

METHOD PUBLIC GetValveRetract : BOOL
GetValveRetract := io.outValveRetract;
END_METHOD

// Map a single permissive bit into advancePermissives so tests can force
// REJECTED_PERMISSIVE_NOT_MET / PermissivesNotOK without touching the
// production code's permissive wiring.
METHOD PUBLIC MapAdvancePerm
VAR_INPUT
    nBit   : UDINT;
    bValue : BOOL;
END_VAR
advancePermissives.MapInput(bitIndex := nBit, inputValue := bValue);
END_METHOD

METHOD PUBLIC MapRetractPerm
VAR_INPUT
    nBit   : UDINT;
    bValue : BOOL;
END_VAR
retractPermissives.MapInput(bitIndex := nBit, inputValue := bValue);
END_METHOD

END_FUNCTION_BLOCK

// ---- POUs/FB_AnalogInput_Probe.TcPOU
// Test-only child of FB_AnalogInput. The production FB keeps its
// hardware-linked `io` UNION in a private VAR section, so tests use this
// probe to inject raw terminal bytes via the UNION alias that matches
// the inputType under test (nInt, fReal, di, ...).
//
// The probe delegates the cyclic body back to the parent via SUPER^()
// so the inherited conditioning pipeline runs against the injected raw
// value. Without that call the child's empty body would replace the
// parent logic and every assertion would see zeroed status.
//
// Lives in the Testing project only — not part of TcForge's public API.
FUNCTION_BLOCK FB_AnalogInput_Probe EXTENDS TcForge.FB_AnalogInput

SUPER^();

// Inject the raw terminal value via the INT alias of the UNION.
// Pair with cfg.inputType := __SYSTEM.TYPE_CLASS.TYPE_INT.
METHOD PUBLIC SetRawInt
VAR_INPUT
    nValue : INT;
END_VAR
io.inRaw.nInt := nValue;
END_METHOD

// Inject the raw terminal value via the REAL alias of the UNION.
// Pair with cfg.inputType := __SYSTEM.TYPE_CLASS.TYPE_REAL.
METHOD PUBLIC SetRawReal
VAR_INPUT
    fValue : REAL;
END_VAR
io.inRaw.fReal := fValue;
END_METHOD

// Inject the raw terminal value via the DINT alias of the UNION.
// Pair with cfg.inputType := __SYSTEM.TYPE_CLASS.TYPE_DINT.
METHOD PUBLIC SetRawDInt
VAR_INPUT
    nValue : DINT;
END_VAR
io.inRaw.di := nValue;
END_METHOD

END_FUNCTION_BLOCK

// ---- POUs/FB_AnalogOutput_Probe.TcPOU
// Test-only child of FB_AnalogOutput. The production FB keeps its
// hardware-linked `io` UNION in a private VAR section, so tests use
// this probe to *read back* whichever UNION member the FB wrote into
// (nInt, fReal, dw, ...). We don't need a writer here because the
// production FB drives the write side via SetValue and the scaling
// pipeline — the tests only need to verify that the correct UNION
// alias actually got the expected bytes.
//
// The probe delegates the cyclic body back to the parent via SUPER^()
// so the inherited pipeline runs. Without that call the child's empty
// body would replace the parent logic and every assertion would see
// zeroed I/O.
//
// Lives in the Testing project only — not part of TcForge's public API.
FUNCTION_BLOCK FB_AnalogOutput_Probe EXTENDS TcForge.FB_AnalogOutput

SUPER^();

// Read back what the FB last wrote to the INT alias of the UNION.
// Pair with cfg.outputType := __SYSTEM.TYPE_CLASS.TYPE_INT.
METHOD PUBLIC GetRawInt : INT
GetRawInt := io.outRaw.nInt;
END_METHOD

// Read back what the FB last wrote to the REAL alias of the UNION.
// Pair with cfg.outputType := __SYSTEM.TYPE_CLASS.TYPE_REAL.
METHOD PUBLIC GetRawReal : REAL
GetRawReal := io.outRaw.fReal;
END_METHOD

// Read back the raw DWORD view of the UNION. Handy for verifying that
// a skipped write (e.g. under BAD quality) really left the previous
// bytes untouched, independent of which alias was last active.
METHOD PUBLIC GetRawDWord : DWORD
GetRawDWord := io.outRaw.dw;
END_METHOD

END_FUNCTION_BLOCK
